// TIA Portal V20 export
TYPE "typeIdentMvHmi"
// stored: Access Published
   STRUCT
      selectedUnit : USInt;
      selectedEM : USInt;
      mvReaderId : USInt;   // MV Reader ID
      numberOfMv : USInt;   // Anzahl der MV Antriebe / Number of used MV readers
      mvReader : Array[0.."NO_OF_MV_IDENT_DEVICES"] of "LSicar_typeIdentInterfaceHmi";   // MV Reader
   END_STRUCT;
END_TYPE
